PROGRAM Move_Command
VAR
	vis_x :  LREAL ;
	vis_y :  LREAL ;
	vis_r :  LREAL ;
	Motor_Move_Trig          : R_TRIG;
END_VAR


vis_x := GVL_Vision.Axis02_Calibration_Position_Data;
vis_y := GVL_Vision.Axis03_Calibration_Position_Data;
vis_r := GVL_Vision.Axis05_Calibration_Position_Data;

Motor_Move_Trig(CLK := GVL_Calibration.Motor_Move);

IF  Motor_Move_Trig.Q THEN
	GVL_Axis02.Calibration_Position := FALSE;
	GVL_Axis03.Calibration_Position := FALSE;
	GVL_Axis05.Calibration_Position := FALSE;
	GVL_Calibration.Calibration_Pos_Moving := TRUE;
END_IF

IF GVL_Axis02.Calibration_Position AND GVL_Axis03.Calibration_Position AND GVL_Axis05.Calibration_Position THEN
	GVL_Calibration.Motor_Move := FALSE;
	GVL_Calibration.Calibration_Pos_Moving := FALSE;
END_IF

END_PROGRAM

(* stored: Version 1.1.0.1, ProductVersion 3.1.4024.15
   POU Move_Command: Id {025a35f5-28d2-4787-834e-1b98fbe85877}, SpecialFunc None *)
